(* Logix 5000 project; controller Process_Output Emulate 5570 rev 33.11; software revision 33.00 *)

TASK MainTask (continuous, watchdog 500 ms) : MainProgram

MODULES
   Local : Emulate 5570 (ICP 2, rev 33.11)
       : 1756-IB16 (ICP 3, rev 3.1, Input RPI 20 ms)
       : vendor 1 type 7 code 16 (ICP 4, rev 3.1, Output RPI 20 ms)
END_MODULES

PROGRAM MainProgram   (* main routine FuncRoutine *)

ROUTINE FuncRoutine   (* function block diagram *)
   SHEET 1
END_ROUTINE
END_PROGRAM
